LIN {X 0,Y 38.072,Z 381.149,A -85,B 0,C 180,E1 -30886.764,E2 -30886.764} C_VEL
LIN {X 0,Y 37.778,Z 378.304,A -85,B 0,C 180,E1 -30891.542,E2 -30891.542} C_VEL
LIN {X 0,Y 37.157,Z 375.673,A -85,B 0,C 180,E1 -30897.217,E2 -30897.217} C_VEL
LIN {X 0,Y 35.861,Z 371.779,A -85,B 0,C 180,E1 -30908.382,E2 -30908.382} C_VEL
LIN {X 0,Y 35.068,Z 369.625,A -85,B 0,C 180,E1 -30918.536,E2 -30918.536} C_VEL
LIN {X 0,Y 34.88,Z 368.932,A -85,B 0,C 180,E1 -30923.704,E2 -30923.704} C_VEL
LIN {X 0,Y 34.921,Z 368.357,A -85,B 0,C 180,E1 -30936.266,E2 -30936.266} C_VEL
LIN {X 0,Y 35.868,Z 369.212,A -85,B 0,C 180,E1 -30948.702,E2 -30948.702} C_VEL
LIN {X 0,Y 36.482,Z 371.166,A -85,B 0,C 180,E1 -30955.874,E2 -30955.874} C_VEL
LIN {X 0,Y 37.236,Z 375.236,A -85,B 0,C 180,E1 -30965.417,E2 -30965.417} C_VEL
LIN {X 0,Y 38.121,Z 379.41,A -85,B 0,C 180,E1 -30973.328,E2 -30973.328} C_VEL
LIN {X 0,Y 38.329,Z 381.079,A -85,B 0,C 180,E1 -30975.971,E2 -30975.971} C_VEL
LIN {X 0,Y 33.947,Z 393.088,A -85,B 0,C 180,E1 -30986.887,E2 -30986.887} C_VEL
LIN {X 0,Y 30.53,Z 402.361,A -85,B 0,C 180,E1 -30999.021,E2 -30999.021} C_VEL
LIN {X 0,Y 29.181,Z 405.342,A -85,B 0,C 180,E1 -31003.736,E2 -31003.736} C_VEL
LIN {X 0,Y 25.277,Z 412.112,A -85,B 0,C 180,E1 -31017.084,E2 -31017.084} C_VEL
LIN {X 0,Y 23.052,Z 415.703,A -85,B 0,C 180,E1 -31026.967,E2 -31026.967} C_VEL
LIN {X 0,Y 20.619,Z 418.794,A -85,B 0,C 180,E1 -31038.764,E2 -31038.764} C_VEL
LIN {X 0,Y 18.019,Z 423.93,A -85,B 0,C 180,E1 -31070.966,E2 -31070.966} C_VEL
LIN {X 0,Y 20.097,Z 426.963,A -85,B 0,C 180,E1 -31092.924,E2 -31092.924} C_VEL
LIN {X 0,Y 26.361,Z 430.594,A -85,B 0,C 180,E1 -31111.083,E2 -31111.083} C_VEL
LIN {X 0,Y 28.434,Z 431.385,A -85,B 0,C 180,E1 -31116.328,E2 -31116.328} C_VEL
LIN {X 0,Y 19.724,Z 425.924,A -85,B 0,C 180,E1 -31132.276,E2 -31132.276} C_VEL
LIN {X 0,Y 14.05,Z 418.42,A -85,B 0,C 180,E1 -31170.009,E2 -31170.009} C_VEL
LIN {X 0,Y 16.611,Z 409.801,A -85,B 0,C 180,E1 -31212.154,E2 -31212.154} C_VEL
LIN {X 0,Y 22.867,Z 401.003,A -85,B 0,C 180,E1 -31232.963,E2 -31232.963} C_VEL
LIN {X 0,Y 29.882,Z 391.377,A -85,B 0,C 180,E1 -31243.603,E2 -31243.603} C_VEL
LIN {X 0,Y 31.837,Z 388.481,A -85,B 0,C 180,E1 -31245.719,E2 -31245.719} C_VEL
LIN {X 0,Y 32.398,Z 386.918,A -85,B 0,C 180,E1 -31247.613,E2 -31247.613} C_VEL
LIN {X 0,Y 32.69,Z 382.628,A -85,B 0,C 180,E1 -31255.466,E2 -31255.466} C_VEL
LIN {X 0,Y 32.47,Z 380.807,A -85,B 0,C 180,E1 -31260.031,E2 -31260.031} C_VEL
LIN {X 0,Y 31.815,Z 377.39,A -85,B 0,C 180,E1 -31271.506,E2 -31271.506} C_VEL
LIN {X 0,Y 31.57,Z 376.139,A -85,B 0,C 180,E1 -31278.1,E2 -31278.1} C_VEL
LIN {X 0,Y 31.5,Z 374.818,A -85,B 0,C 180,E1 -31293.501,E2 -31293.501} C_VEL
LIN {X 0,Y 32.272,Z 375.485,A -85,B 0,C 180,E1 -31307.423,E2 -31307.423} C_VEL
LIN {X 0,Y 32.548,Z 377.721,A -85,B 0,C 180,E1 -31315.374,E2 -31315.374} C_VEL
LIN {X 0,Y 32.852,Z 382.474,A -85,B 0,C 180,E1 -31326.913,E2 -31326.913} C_VEL
LIN {X 0,Y 32.726,Z 383.868,A -85,B 0,C 180,E1 -31329.27,E2 -31329.27} C_VEL
LIN {X 0,Y 27.393,Z 395.436,A -85,B 0,C 180,E1 -31341.557,E2 -31341.557} C_VEL
LIN {X 0,Y 24.001,Z 402.677,A -85,B 0,C 180,E1 -31353.049,E2 -31353.049} C_VEL
LIN {X 0,Y 20.762,Z 407.58,A -85,B 0,C 180,E1 -31362.613,E2 -31362.613} C_VEL
LIN {X 0,Y 16.267,Z 416.028,A -85,B 0,C 180,E1 -31391.093,E2 -31391.093} C_VEL
LIN {X 0,Y 16.686,Z 422.064,A -85,B 0,C 180,E1 -31422.158,E2 -31422.158} C_VEL
LIN {X 0,Y 17.662,Z 424.027,A -85,B 0,C 180,E1 -31433.448,E2 -31433.448} C_VEL
LIN {X 0,Y 20.097,Z 426.963,A -85,B 0,C 180,E1 -31452.924,E2 -31452.924} C_VEL
LIN {X 0,Y 20.151,Z 427.158,A -85,B 0,C 180,E1 -31456.588,E2 -31456.588} C_VEL
LIN {X 0,Y 18.998,Z 426.653,A -85,B 0,C 180,E1 -31462.775,E2 -31462.775} C_VEL
LIN {X 0,Y 16.562,Z 425.216,A -85,B 0,C 180,E1 -31470.432,E2 -31470.432} C_VEL
LIN {X 0,Y 10.636,Z 420.897,A -85,B 0,C 180,E1 -31488.734,E2 -31488.734} C_VEL
LIN {X 0,Y 7.258,Z 416.792,A -85,B 0,C 180,E1 -31521.53,E2 -31521.53} C_VEL
LIN {X 0,Y 11.071,Z 408.163,A -85,B 0,C 180,E1 -31589.999,E2 -31589.999} C_VEL
LIN {X 0,Y 18.716,Z 399.474,A -85,B 0,C 180,E1 -31608.463,E2 -31608.463} C_VEL
LIN {X 0,Y 25.975,Z 390.437,A -85,B 0,C 180,E1 -31615.663,E2 -31615.663} C_VEL
LIN {X 0,Y 27.2,Z 388.7,A -85,B 0,C 180,E1 -31616.665,E2 -31616.665} C_VEL
LIN {X 0,Y 27.576,Z 386.889,A -85,B 0,C 180,E1 -31620.645,E2 -31620.645} C_VEL
LIN {X 0,Y 27.654,Z 385.156,A -85,B 0,C 180,E1 -31625.989,E2 -31625.989} C_VEL
LIN {X 0,Y 27.697,Z 382.152,A -85,B 0,C 180,E1 -31639.574,E2 -31639.574} C_VEL
LIN {X 0,Y 27.682,Z 381.375,A -85,B 0,C 180,E1 -31649.487,E2 -31649.487} C_VEL
LIN {X 0,Y 28.403,Z 381.504,A -85,B 0,C 180,E1 -31665.676,E2 -31665.676} C_VEL
LIN {X 0,Y 28.047,Z 384.327,A -85,B 0,C 180,E1 -31675.016,E2 -31675.016} C_VEL
LIN {X 0,Y 27.978,Z 385.191,A -85,B 0,C 180,E1 -31677.505,E2 -31677.505} C_VEL
LIN {X 0,Y 27.635,Z 386.493,A -85,B 0,C 180,E1 -31680.002,E2 -31680.002} C_VEL
LIN {X 0,Y 21.544,Z 397.052,A -85,B 0,C 180,E1 -31691.864,E2 -31691.864} C_VEL
LIN {X 0,Y 17.47,Z 403.516,A -85,B 0,C 180,E1 -31703.724,E2 -31703.724} C_VEL
LIN {X 0,Y 10.023,Z 413.158,A -85,B 0,C 180,E1 -31738.273,E2 -31738.273} C_VEL
LIN {X 0,Y 10.11,Z 419.532,A -85,B 0,C 180,E1 -31790.341,E2 -31790.341} C_VEL
LIN {X 0,Y 11.78,Z 421.613,A -85,B 0,C 180,E1 -31806.628,E2 -31806.628} C_VEL
LIN {X 0,Y 16.104,Z 424.923,A -85,B 0,C 180,E1 -31830.789,E2 -31830.789} C_VEL
LIN {X 0,Y 15.68,Z 424.611,A -85,B 0,C 180,E1 -31833.693,E2 -31833.693} C_VEL
LIN {X 0,Y 7.258,Z 416.792,A -85,B 0,C 180,E1 -31881.53,E2 -31881.53} C_VEL
LIN {X 0,Y 6.755,Z 414.418,A -85,B 0,C 180,E1 -31906.895,E2 -31906.895} C_VEL
LIN {X 0,Y 7.533,Z 410.591,A -85,B 0,C 180,E1 -31943.189,E2 -31943.189} C_VEL
LIN {X 0,Y 14.25,Z 400.782,A -85,B 0,C 180,E1 -31985.215,E2 -31985.215} C_VEL
LIN {X 0,Y 17.977,Z 396.266,A -85,B 0,C 180,E1 -31989.916,E2 -31989.916} C_VEL
LIN {X 0,Y 19.258,Z 394.737,A -85,B 0,C 180,E1 -31990.342,E2 -31990.342} C_VEL
LIN {X 0,Y 22.96,Z 390.105,A -85,B 0,C 180,E1 -31991.3,E2 -31991.3} C_VEL
LIN {X 0,Y 23.581,Z 387.803,A -85,B 0,C 180,E1 -32003.414,E2 -32003.414} C_VEL
LIN {X 0,Y 23.74,Z 387.295,A -85,B 0,C 180,E1 -32012.64,E2 -32012.64} C_VEL
LIN {X 0,Y 24.098,Z 387.486,A -85,B 0,C 180,E1 -32023.046,E2 -32023.046} C_VEL
LIN {X 0,Y 23.696,Z 388.527,A -85,B 0,C 180,E1 -32026.718,E2 -32026.718} C_VEL
LIN {X 0,Y 16.461,Z 398.668,A -85,B 0,C 180,E1 -32036.347,E2 -32036.347} C_VEL
LIN {X 0,Y 14.058,Z 401.727,A -85,B 0,C 180,E1 -32041.05,E2 -32041.05} C_VEL
LIN {X 0,Y 7.155,Z 408.504,A -85,B 0,C 180,E1 -32050.795,E2 -32050.795} C_VEL
LIN {X 0,Y 2.221,Z 414.229,A -85,B 0,C 180,E1 -32130.003,E2 -32130.003} C_VEL
LIN {X 0,Y 0.128,Z 413.224,A -85,B 0,C 180,E1 -32309.954,E2 -32309.954} C_VEL
LIN {X 0,Y 10.326,Z 404.336,A -85,B 0,C 180,E1 -32348.95,E2 -32348.95} C_VEL
LIN {X 0,Y 19.258,Z 394.737,A -85,B 0,C 180,E1 -32350.342,E2 -32350.342} C_VEL
LIN {X 0,Y 22.785,Z 396.025,A -85,B 0,C 180,E1 -32350.731,E2 -32350.731} C_VEL
LIN {X 0,Y 22.785,Z 600,A -85,B 0,C 180,E1 -32350.731,E2 -32350.731} C_VEL
LIN {X 0,Y 22.785,Z 600,A -85,B 0,C 180,E1 -32350.731,E2 -32350.731}

QRS_NEXT_CUT()

QRS_NEXT()
QRS_HOME()

END
